FUNCTION_BLOCK FB_CalcFocalLengthSingleLensMock EXTENDS FB_FalliblePublicMock IMPLEMENTS I_CalcFocalLengthSingleLens
VAR
    fbFocalLength : FB_QuantityLREALPublic(Units := 'm');
    afFocalLength : ARRAY[1..GVL_Physics.nMaxNumLensesInSet] OF LREAL;
    nIndex : INT;
END_VAR


METHOD Calculate
VAR_INPUT
    Lens : I_Lens;
END_VAR
VAR_IN_OUT
    FocalLength : FB_QuantityLREALPublic(Units := 'm');
END_VAR

nIndex := nIndex + 1;

IF nIndex > GVL_Physics.nMaxNumLensesInSet THEN
    nIndex := 1;
END_IF

fbFocalLength.Val := afFocalLength[nIndex];

FocalLength := fbFocalLength;
END_METHOD


METHOD SetResult
VAR_INPUT
    Result : LREAL;
    LensNum : INT;
END_VAR

afFocalLength[LensNum] := Result;
END_METHOD


METHOD SetValid

fbFocalLength.Val := 1.0;
fbFocalLength.Units := 'm';
fbFocalLength.ClearError();
ClearError();

FOR nIndex := 1 TO GVL_Physics.nMaxNumLensesInSet DO
    afFocalLength[nIndex] := 1.0;
END_FOR
END_METHOD

END_FUNCTION_BLOCK

(* stored: Version 1.1.0.1
   POU FB_CalcFocalLengthSingleLensMock: Id {6906ef4b-70f5-42bd-b512-b76eb2dac2e2}, SpecialFunc None
   Method Calculate: Id {b2c83659-42d3-4010-bd66-b5ff217644cd}
   Method SetResult: Id {fa56926d-e362-4a57-9807-06847d87b563}
   Method SetValid: Id {dad76da5-b9b0-428c-86cd-6f3a241cdfd8} *)
